Omron CX-Programmer project NewProject (CX-Programmer 9.75)

# PLC project02: CP2E-N N

## Program NewProgram1 (cyclic task 0)

### Section Section1

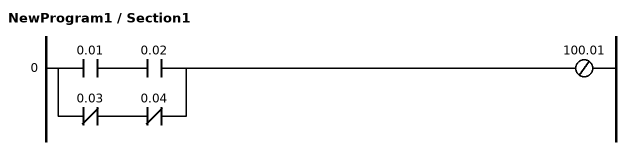
; rung 0
LD 0.01
AND 0.02
LDNOT 0.03
ANDNOT 0.04
ORLD
OUTNOT 100.01

### Section END
; rung 0
END(001)